FUNCTION_BLOCK OPTIMIZE_ENERGY
  {SET_ATTRIBUTE(OpcUa, SERVICE)}
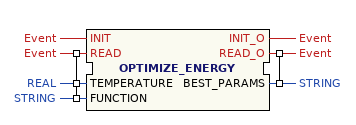
  EVENT_INPUT
    INIT;
    READ WITH TEMPERATURE, FUNCTION;
  END_EVENT
  EVENT_OUTPUT
    INIT_O;
    READ_O WITH BEST_PARAMS;
  END_EVENT
  VAR_INPUT
    TEMPERATURE : REAL; {SET_ATTRIBUTE(OpcUa, Constant)}
    FUNCTION : STRING; {SET_ATTRIBUTE(OpcUa, Variable)}
  END_VAR
  VAR_OUTPUT
    BEST_PARAMS : STRING; {SET_ATTRIBUTE(OpcUa, Variable)}
  END_VAR
END_FUNCTION_BLOCK
